TYPE "Val"
VERSION : 0.1
   STRUCT
      "[Int]" : Int;
      "[Real]" : Real;
      Perc : Int;
   END_STRUCT;

END_TYPE

